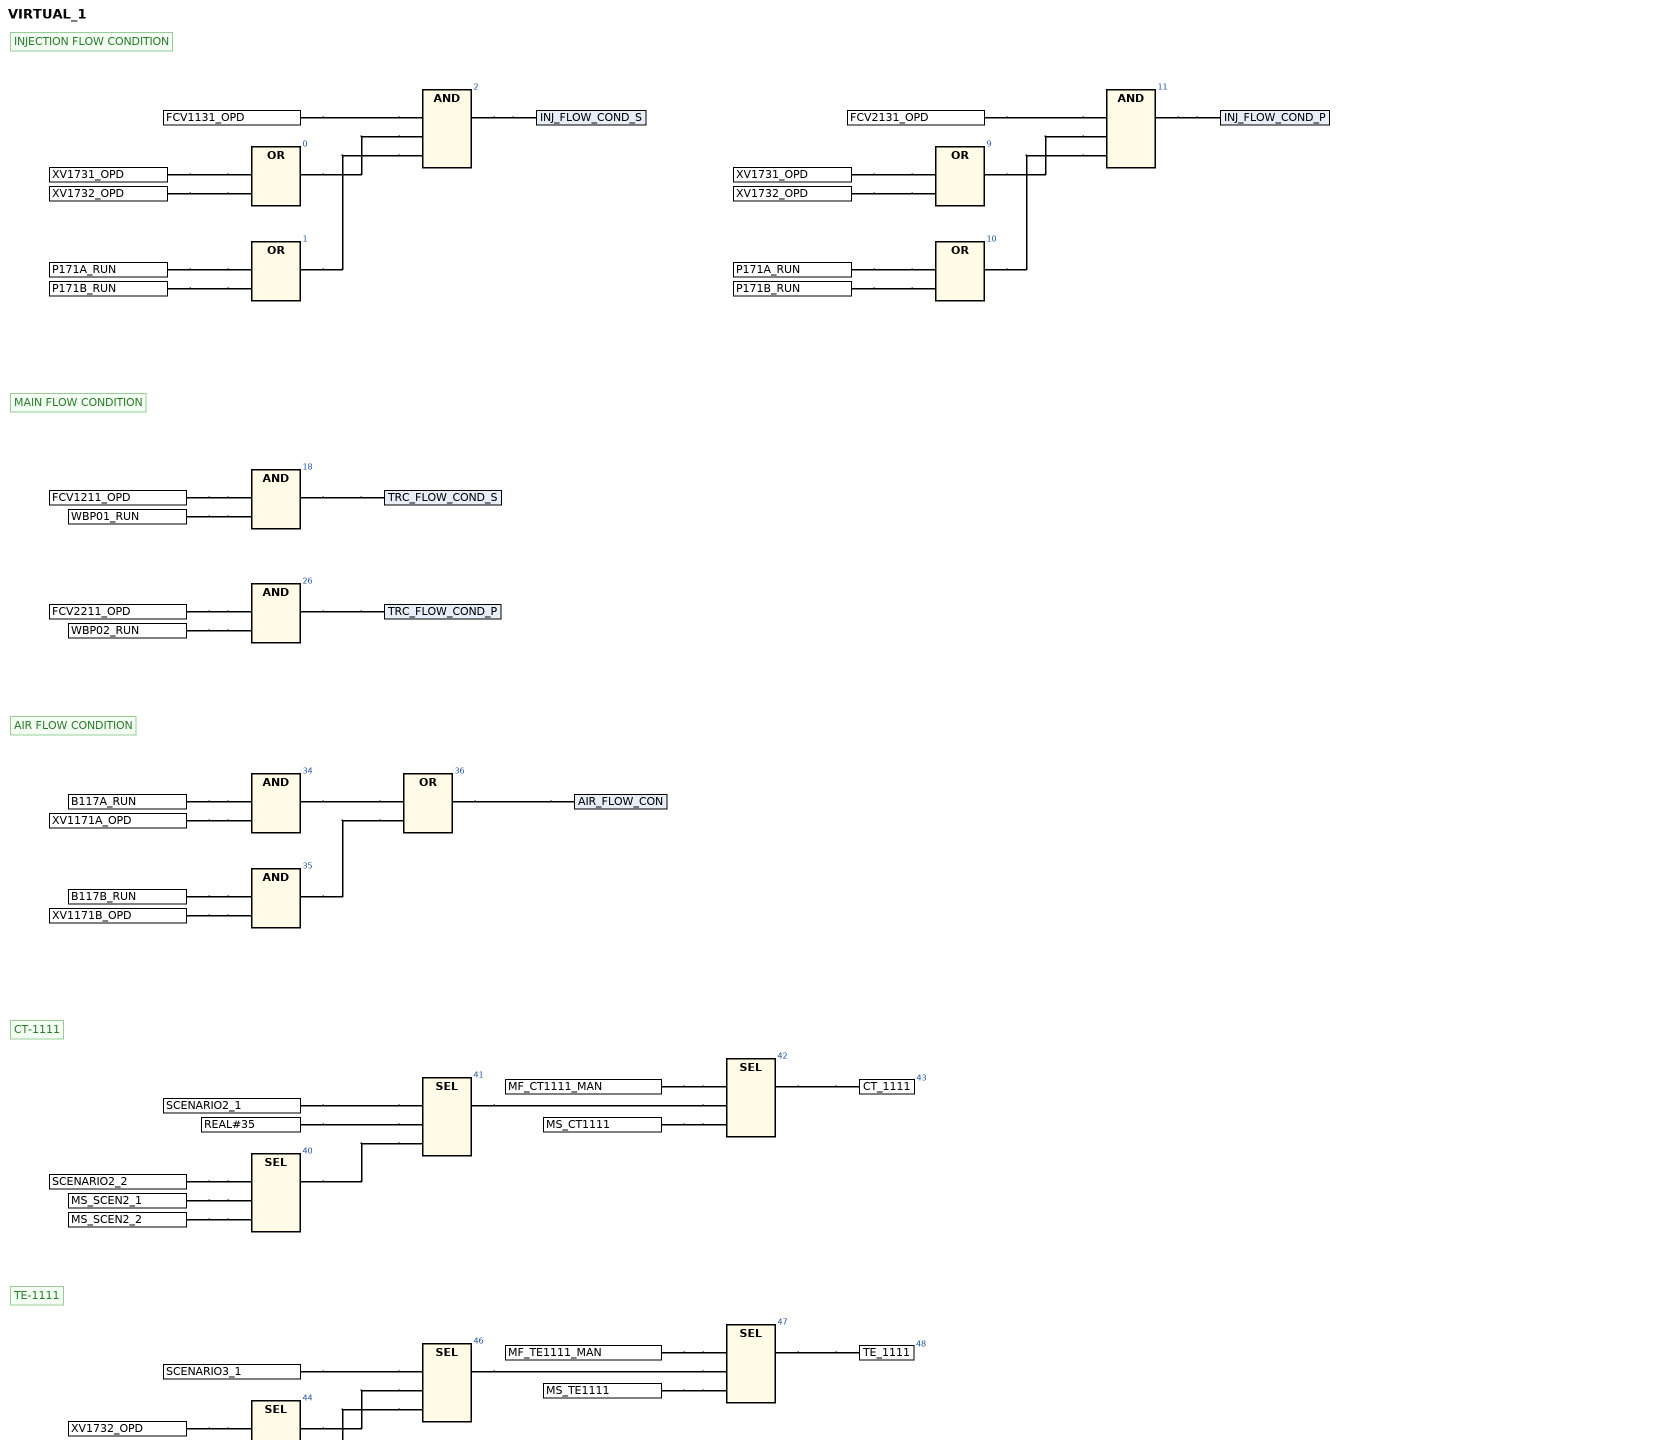
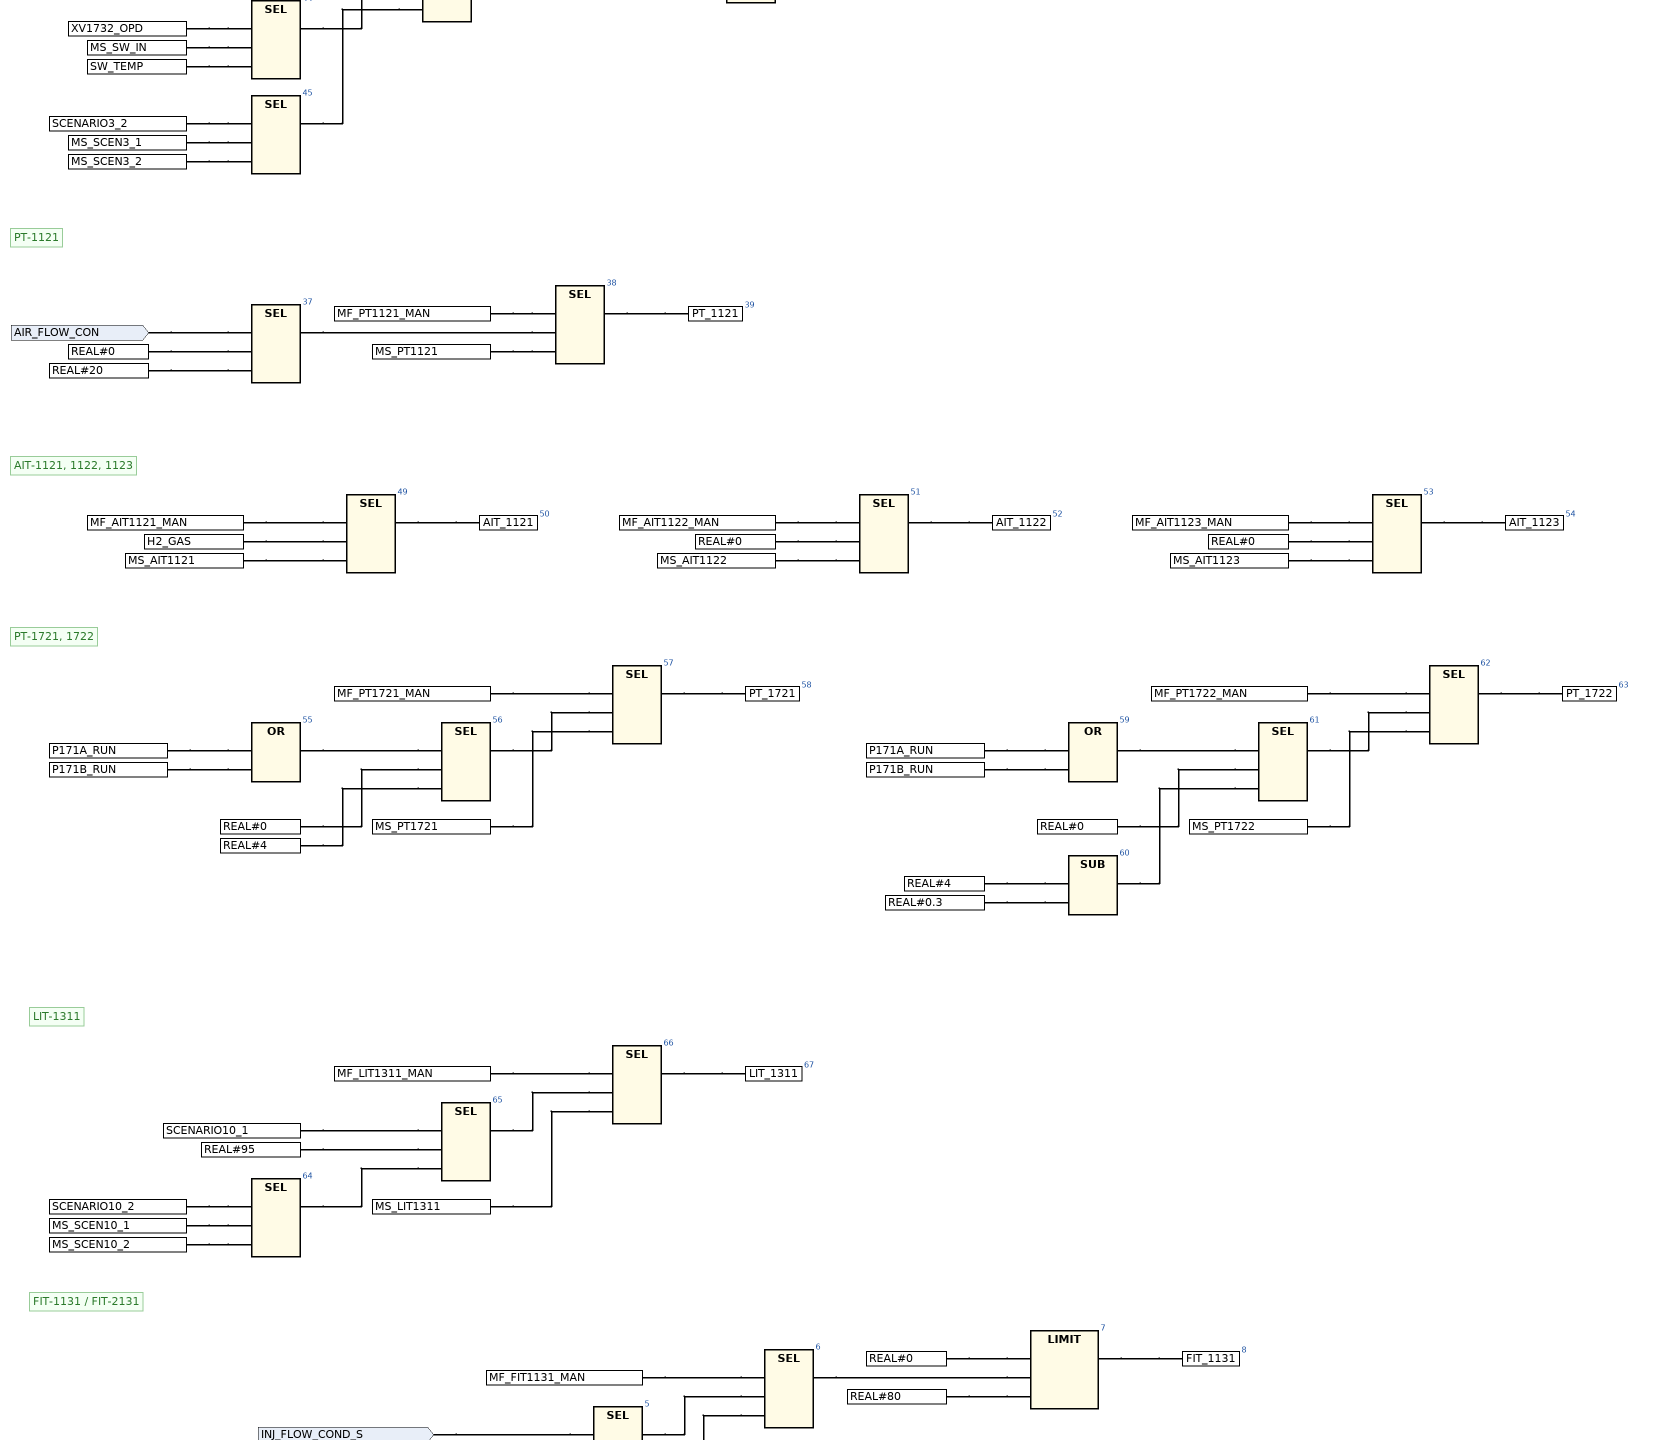
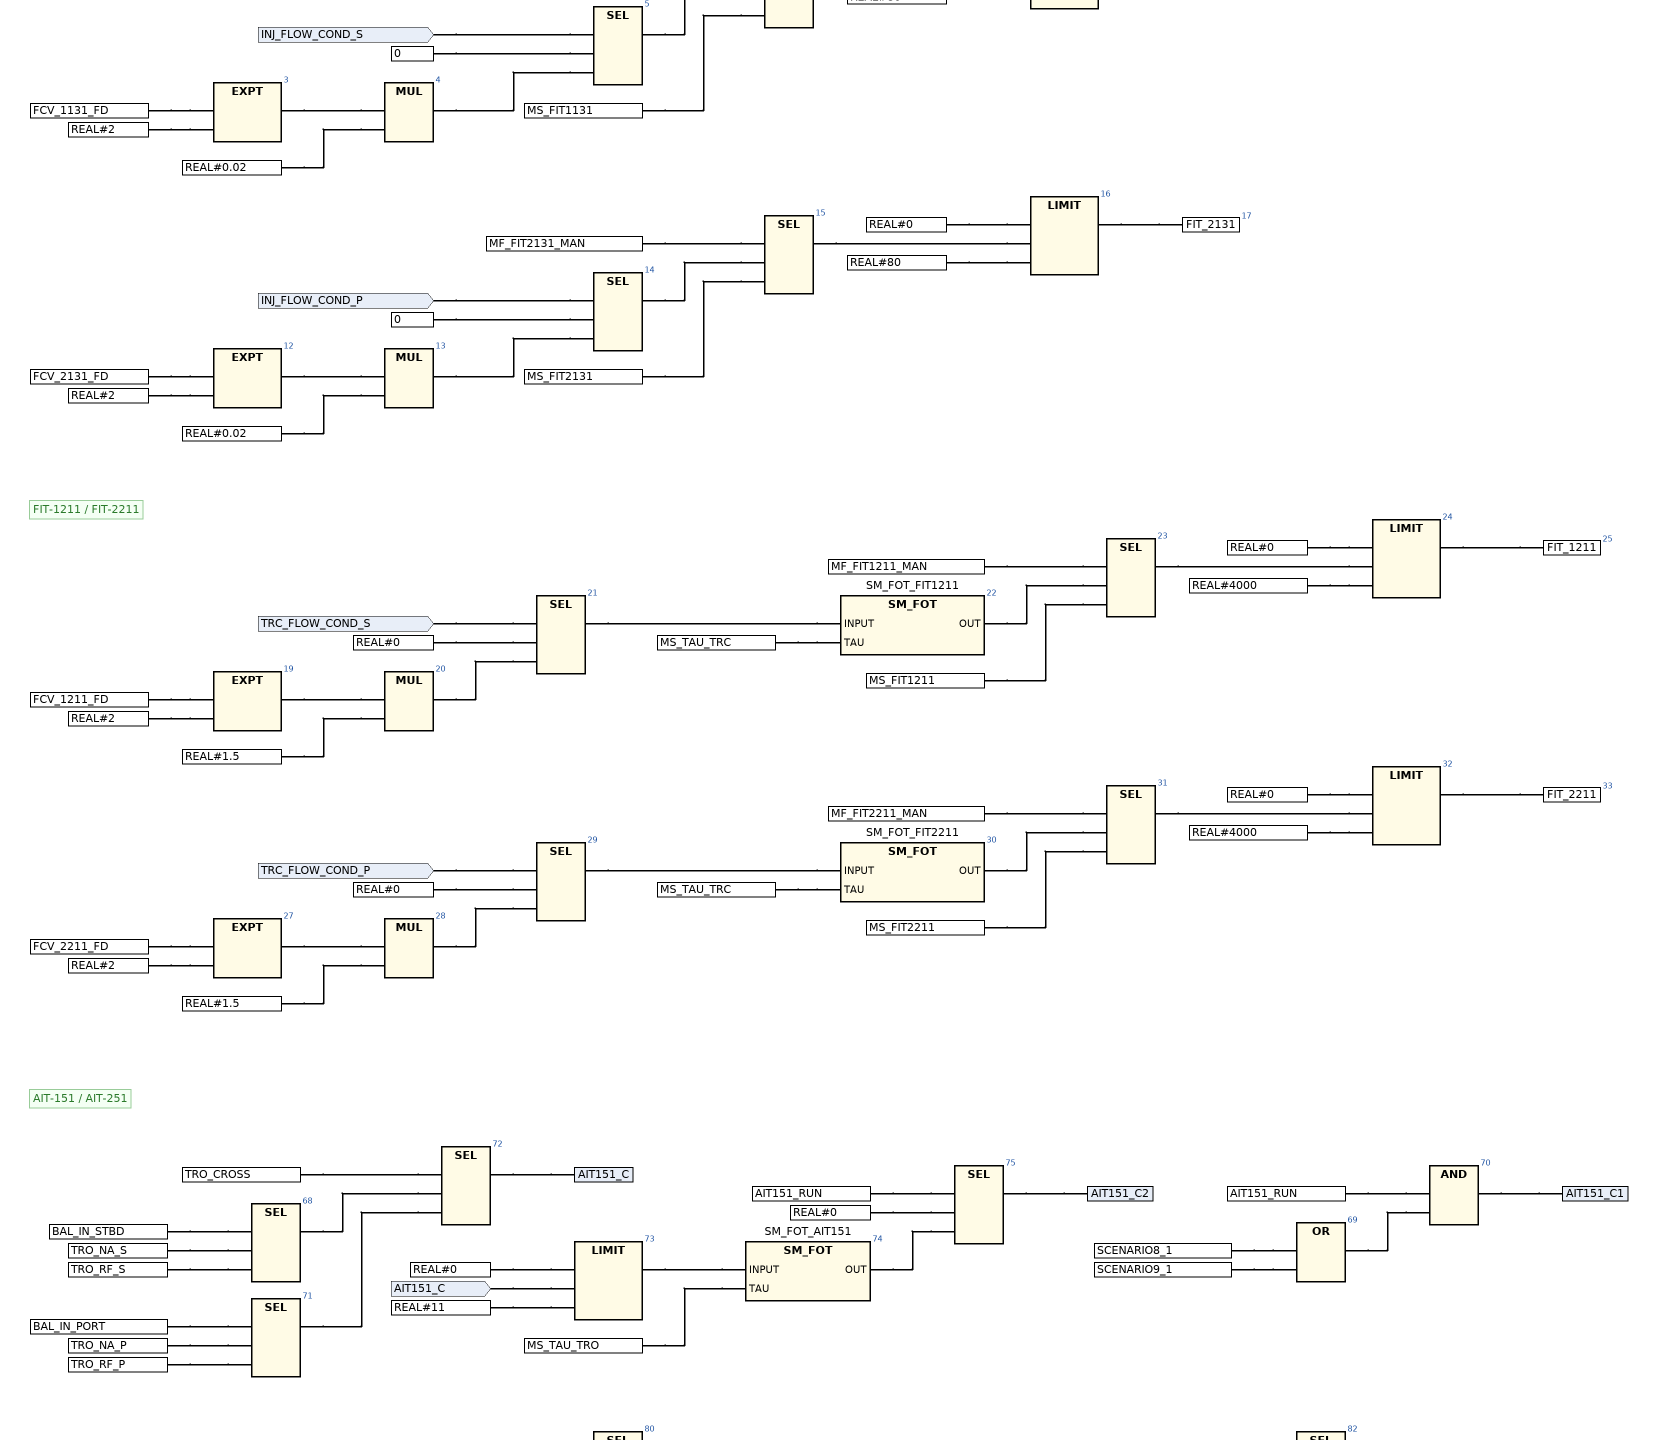
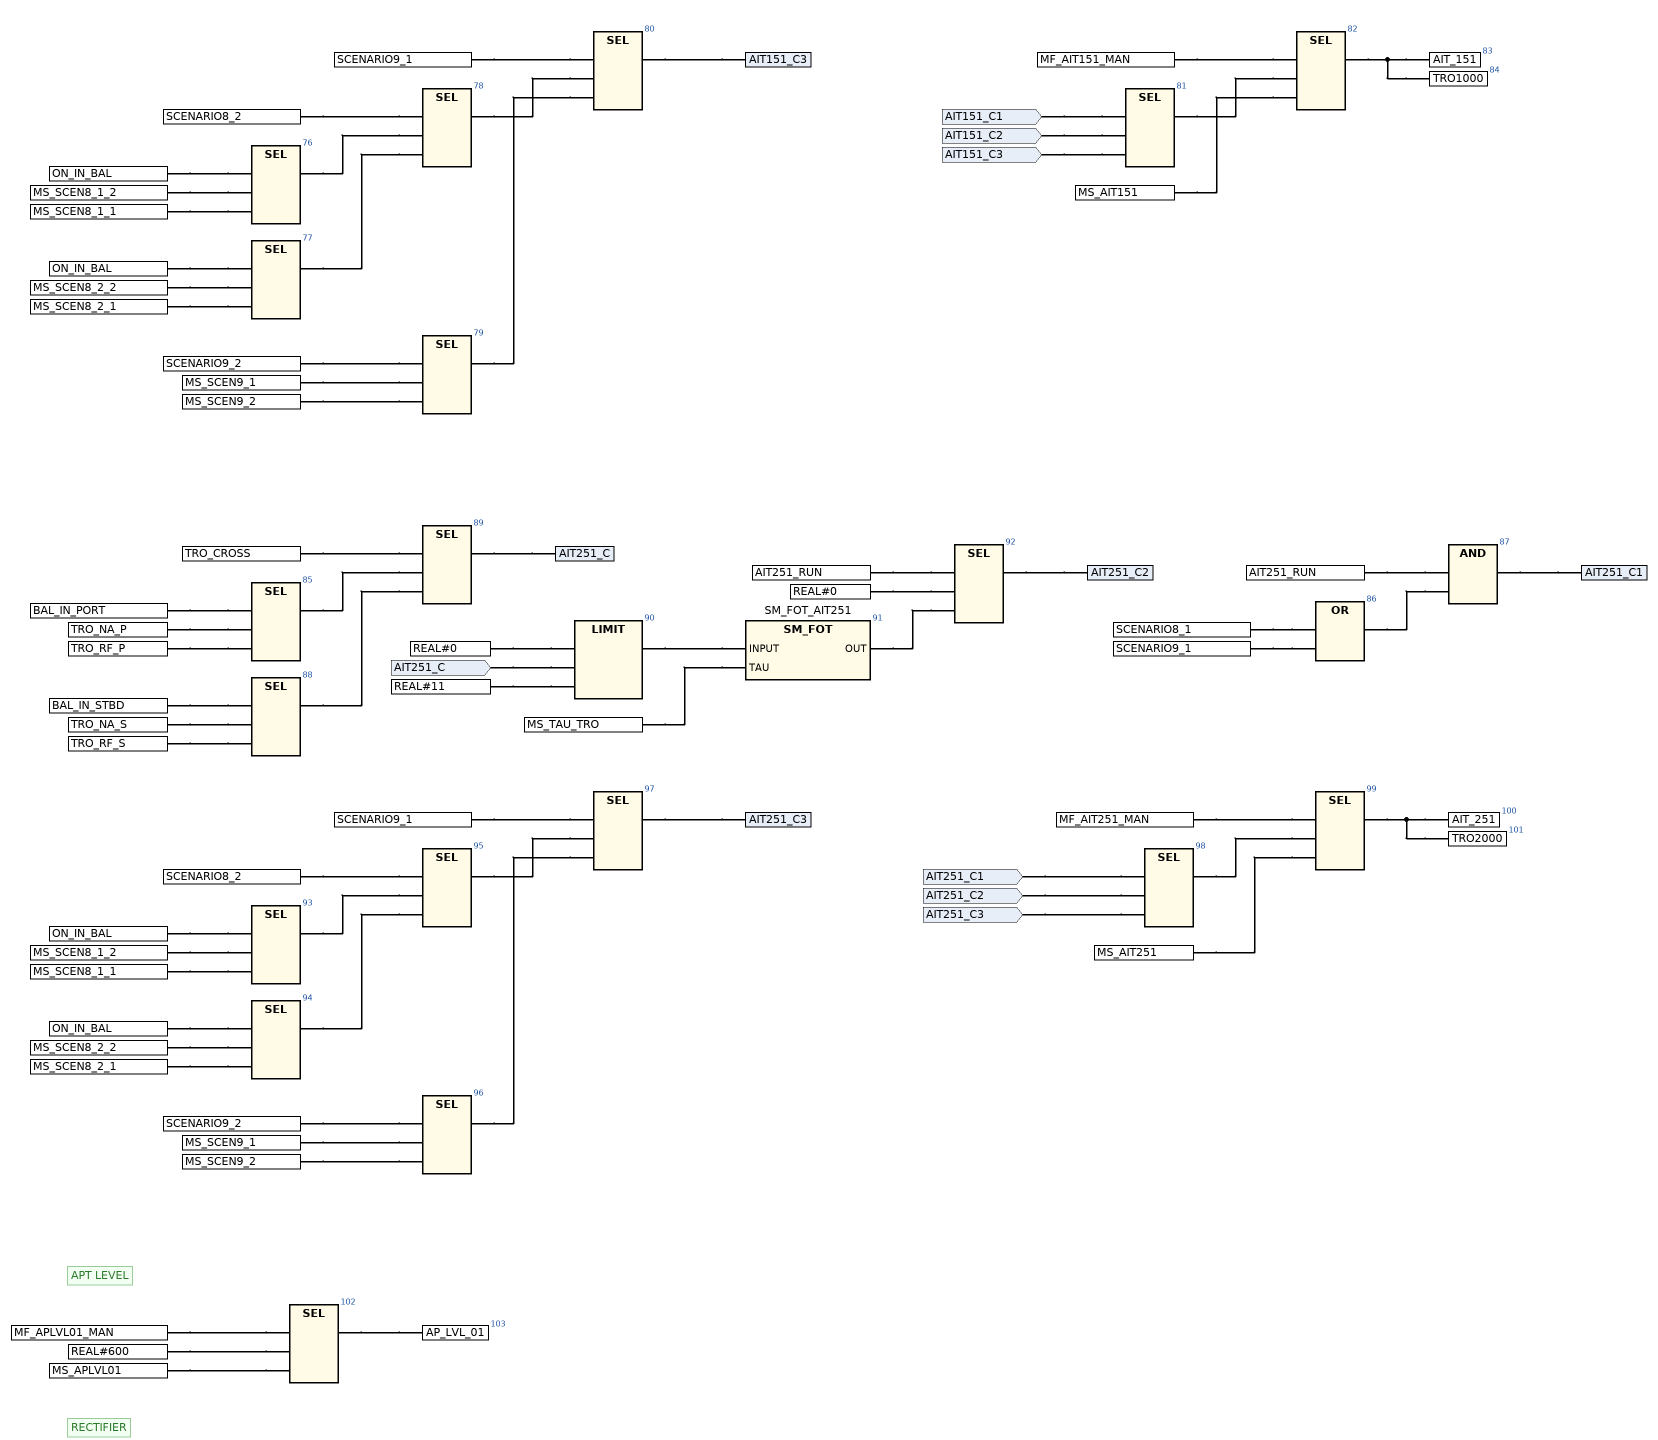
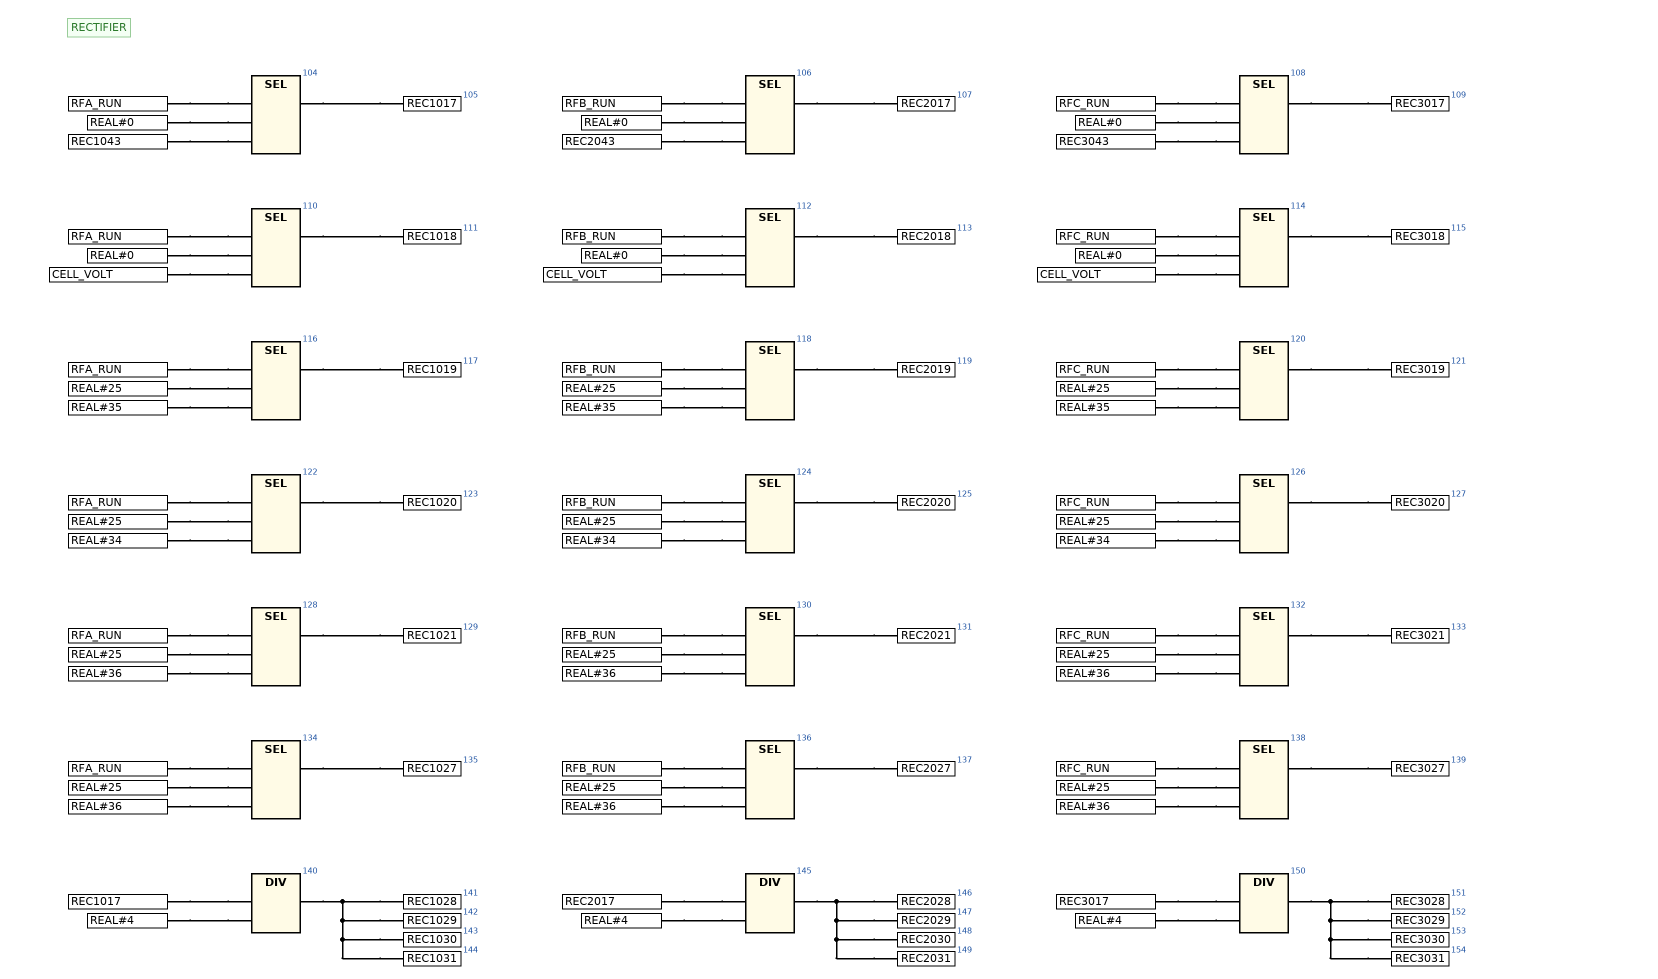
// INJECTION FLOW CONDITION
(* FCV1131_OPD AND (XV1731_OPD OR XV1732_OPD) AND (P171A_RUN OR P171B_RUN); result not used *)
// FIT-1131 / FIT-2131
FIT_1131 := LIMIT(REAL#0, SEL(MF_FIT1131_MAN, SEL(_w1, 0, EXPT(FCV_1131_FD, REAL#2) * REAL#0.02), MS_FIT1131), REAL#80);
(* FCV2131_OPD AND (XV1731_OPD OR XV1732_OPD) AND (P171A_RUN OR P171B_RUN); result not used *)
FIT_2131 := LIMIT(REAL#0, SEL(MF_FIT2131_MAN, SEL(_w2, 0, EXPT(FCV_2131_FD, REAL#2) * REAL#0.02), MS_FIT2131), REAL#80);
// MAIN FLOW CONDITION
(* FCV1211_OPD AND WBP01_RUN; result not used *)
// FIT-1211 / FIT-2211
SM_FOT_FIT1211(INPUT := SEL(_w3, REAL#0, EXPT(FCV_1211_FD, REAL#2) * REAL#1.5), TAU := MS_TAU_TRC); // SM_FOT
FIT_1211 := LIMIT(REAL#0, SEL(MF_FIT1211_MAN, SM_FOT_FIT1211.OUT, MS_FIT1211), REAL#4000);
(* FCV2211_OPD AND WBP02_RUN; result not used *)
SM_FOT_FIT2211(INPUT := SEL(_w4, REAL#0, EXPT(FCV_2211_FD, REAL#2) * REAL#1.5), TAU := MS_TAU_TRC); // SM_FOT
FIT_2211 := LIMIT(REAL#0, SEL(MF_FIT2211_MAN, SM_FOT_FIT2211.OUT, MS_FIT2211), REAL#4000);
// AIR FLOW CONDITION
(* B117A_RUN AND XV1171A_OPD OR B117B_RUN AND XV1171B_OPD; result not used *)
// PT-1121
PT_1121 := SEL(MF_PT1121_MAN, SEL(_w5, REAL#0, REAL#20), MS_PT1121);
// CT-1111
CT_1111 := SEL(MF_CT1111_MAN, SEL(SCENARIO2_1, REAL#35, SEL(SCENARIO2_2, MS_SCEN2_1, MS_SCEN2_2)), MS_CT1111);
// TE-1111
TE_1111 := SEL(MF_TE1111_MAN, SEL(SCENARIO3_1, SEL(XV1732_OPD, MS_SW_IN, SW_TEMP), SEL(SCENARIO3_2, MS_SCEN3_1, MS_SCEN3_2)), MS_TE1111);
// AIT-1121, 1122, 1123
AIT_1121 := SEL(MF_AIT1121_MAN, H2_GAS, MS_AIT1121);
AIT_1122 := SEL(MF_AIT1122_MAN, REAL#0, MS_AIT1122);
AIT_1123 := SEL(MF_AIT1123_MAN, REAL#0, MS_AIT1123);
// PT-1721, 1722
PT_1721 := SEL(MF_PT1721_MAN, SEL(P171A_RUN OR P171B_RUN, REAL#0, REAL#4), MS_PT1721);
PT_1722 := SEL(MF_PT1722_MAN, SEL(P171A_RUN OR P171B_RUN, REAL#0, REAL#4 - REAL#0.3), MS_PT1722);
// LIT-1311
LIT_1311 := SEL(MF_LIT1311_MAN, SEL(SCENARIO10_1, REAL#95, SEL(SCENARIO10_2, MS_SCEN10_1, MS_SCEN10_2)), MS_LIT1311);
// AIT-151 / AIT-251
(* AIT151_RUN AND (SCENARIO8_1 OR SCENARIO9_1); result not used *)
(* SEL(TRO_CROSS, SEL(BAL_IN_STBD, TRO_NA_S, TRO_RF_S), SEL(BAL_IN_PORT, TRO_NA_P, TRO_RF_P)); result not used *)
SM_FOT_AIT151(INPUT := LIMIT(REAL#0, _w6, REAL#11), TAU := MS_TAU_TRO); // SM_FOT
(* SEL(AIT151_RUN, REAL#0, SM_FOT_AIT151.OUT); result not used *)
(* SEL(SCENARIO9_1, SEL(SCENARIO8_2, SEL(ON_IN_BAL, MS_SCEN8_1_2, MS_SCEN8_1_1), SEL(ON_IN_BAL, MS_SCEN8_2_2, MS_SCEN8_2_1)), SEL(SCENARIO9_2, MS_SCEN9_1, MS_SCEN9_2)); result not used *)
_w10 := SEL(MF_AIT151_MAN, SEL(_w7, _w8, _w9), MS_AIT151);
AIT_151 := _w10;
TRO1000 := _w10;
(* AIT251_RUN AND (SCENARIO8_1 OR SCENARIO9_1); result not used *)
(* SEL(TRO_CROSS, SEL(BAL_IN_PORT, TRO_NA_P, TRO_RF_P), SEL(BAL_IN_STBD, TRO_NA_S, TRO_RF_S)); result not used *)
SM_FOT_AIT251(INPUT := LIMIT(REAL#0, _w11, REAL#11), TAU := MS_TAU_TRO); // SM_FOT
(* SEL(AIT251_RUN, REAL#0, SM_FOT_AIT251.OUT); result not used *)
(* SEL(SCENARIO9_1, SEL(SCENARIO8_2, SEL(ON_IN_BAL, MS_SCEN8_1_2, MS_SCEN8_1_1), SEL(ON_IN_BAL, MS_SCEN8_2_2, MS_SCEN8_2_1)), SEL(SCENARIO9_2, MS_SCEN9_1, MS_SCEN9_2)); result not used *)
_w15 := SEL(MF_AIT251_MAN, SEL(_w12, _w13, _w14), MS_AIT251);
AIT_251 := _w15;
TRO2000 := _w15;
// APT LEVEL
AP_LVL_01 := SEL(MF_APLVL01_MAN, REAL#600, MS_APLVL01);
// RECTIFIER
REC1017 := SEL(RFA_RUN, REAL#0, REC1043);
REC2017 := SEL(RFB_RUN, REAL#0, REC2043);
REC3017 := SEL(RFC_RUN, REAL#0, REC3043);
REC1018 := SEL(RFA_RUN, REAL#0, CELL_VOLT);
REC2018 := SEL(RFB_RUN, REAL#0, CELL_VOLT);
REC3018 := SEL(RFC_RUN, REAL#0, CELL_VOLT);
REC1019 := SEL(RFA_RUN, REAL#25, REAL#35);
REC2019 := SEL(RFB_RUN, REAL#25, REAL#35);
REC3019 := SEL(RFC_RUN, REAL#25, REAL#35);
REC1020 := SEL(RFA_RUN, REAL#25, REAL#34);
REC2020 := SEL(RFB_RUN, REAL#25, REAL#34);
REC3020 := SEL(RFC_RUN, REAL#25, REAL#34);
REC1021 := SEL(RFA_RUN, REAL#25, REAL#36);
REC2021 := SEL(RFB_RUN, REAL#25, REAL#36);
REC3021 := SEL(RFC_RUN, REAL#25, REAL#36);
REC1027 := SEL(RFA_RUN, REAL#25, REAL#36);
REC2027 := SEL(RFB_RUN, REAL#25, REAL#36);
REC3027 := SEL(RFC_RUN, REAL#25, REAL#36);
_w16 := REC1017 / REAL#4;
REC1028 := _w16;
REC1029 := _w16;
REC1030 := _w16;
REC1031 := _w16;
_w17 := REC2017 / REAL#4;
REC2028 := _w17;
REC2029 := _w17;
REC2030 := _w17;
REC2031 := _w17;
_w18 := REC3017 / REAL#4;
REC3028 := _w18;
REC3029 := _w18;
REC3030 := _w18;
REC3031 := _w18;

END_PROGRAM

// Device/Application/Logic/0.SIMULATION FBD/SM_FOT
FUNCTION_BLOCK SM_FOT
VAR_INPUT
	INPUT : REAL;
	TAU : REAL := 0.5;				// TIME CONSTANT (0~1)
END_VAR
VAR_OUTPUT
	OUT : REAL;
END_VAR
VAR
	Y1 : REAL;				//EXISTING VALUE
	Y2 : REAL;				//VALUE AFTER CHANGE
	ET_0 : TON;				//ELAPSED TIME AFTER VALUE CHANGE
	INTEGRAL_ET: INTEGRAL;
	TP_0: TP;
END_VAR
VAR // added by the converter: edge detectors and wires of the graphical bodies
    _w1, _w6 : REAL;
    _w2, _w5 : BOOL;
    _w3, _w4, _w7, _w8 : ANY;
END_VAR

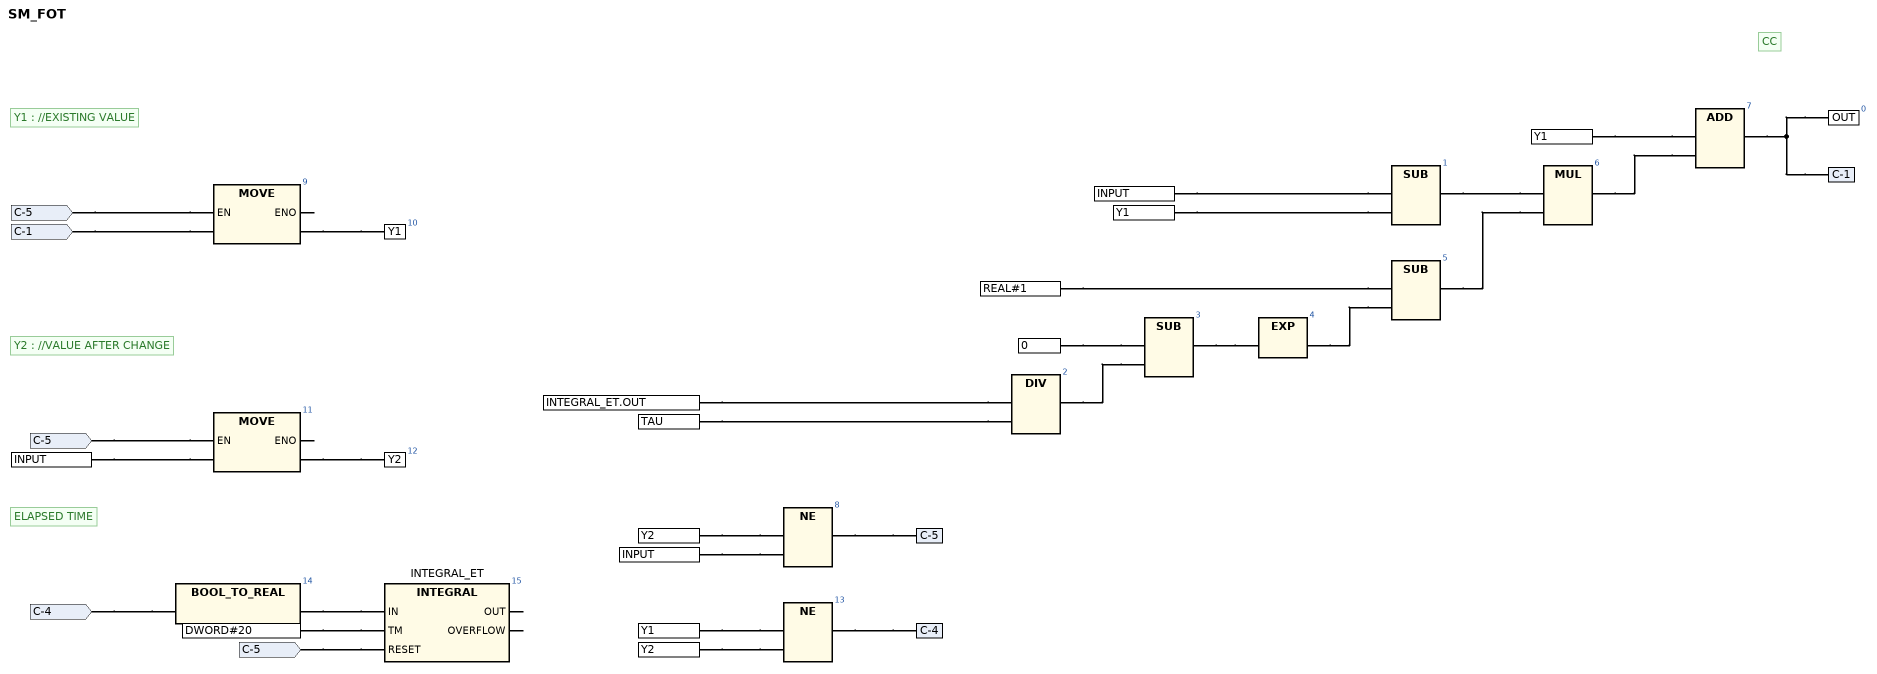
OUT := _w1;
// CC
_w1 := Y1 + (INPUT - Y1) * (REAL#1 - EXP(0 - INTEGRAL_ET.OUT / TAU));
(* Y2 <> INPUT; result not used *)
// Y1 : //EXISTING VALUE
IF _w2 THEN _w4 := _w3; END_IF
Y1 := _w4;
// Y2 : //VALUE AFTER CHANGE
IF _w5 THEN _w6 := INPUT; END_IF
Y2 := _w6;
(* Y1 <> Y2; result not used *)
// ELAPSED TIME
INTEGRAL_ET(IN := BOOL_TO_REAL(_w7), TM := DWORD#20, RESET := _w8); // INTEGRAL

END_FUNCTION_BLOCK

// Device/Application/Logic/0.SIMULATION/VIRTUAL_2
PROGRAM VIRTUAL_2
VAR
END_VAR

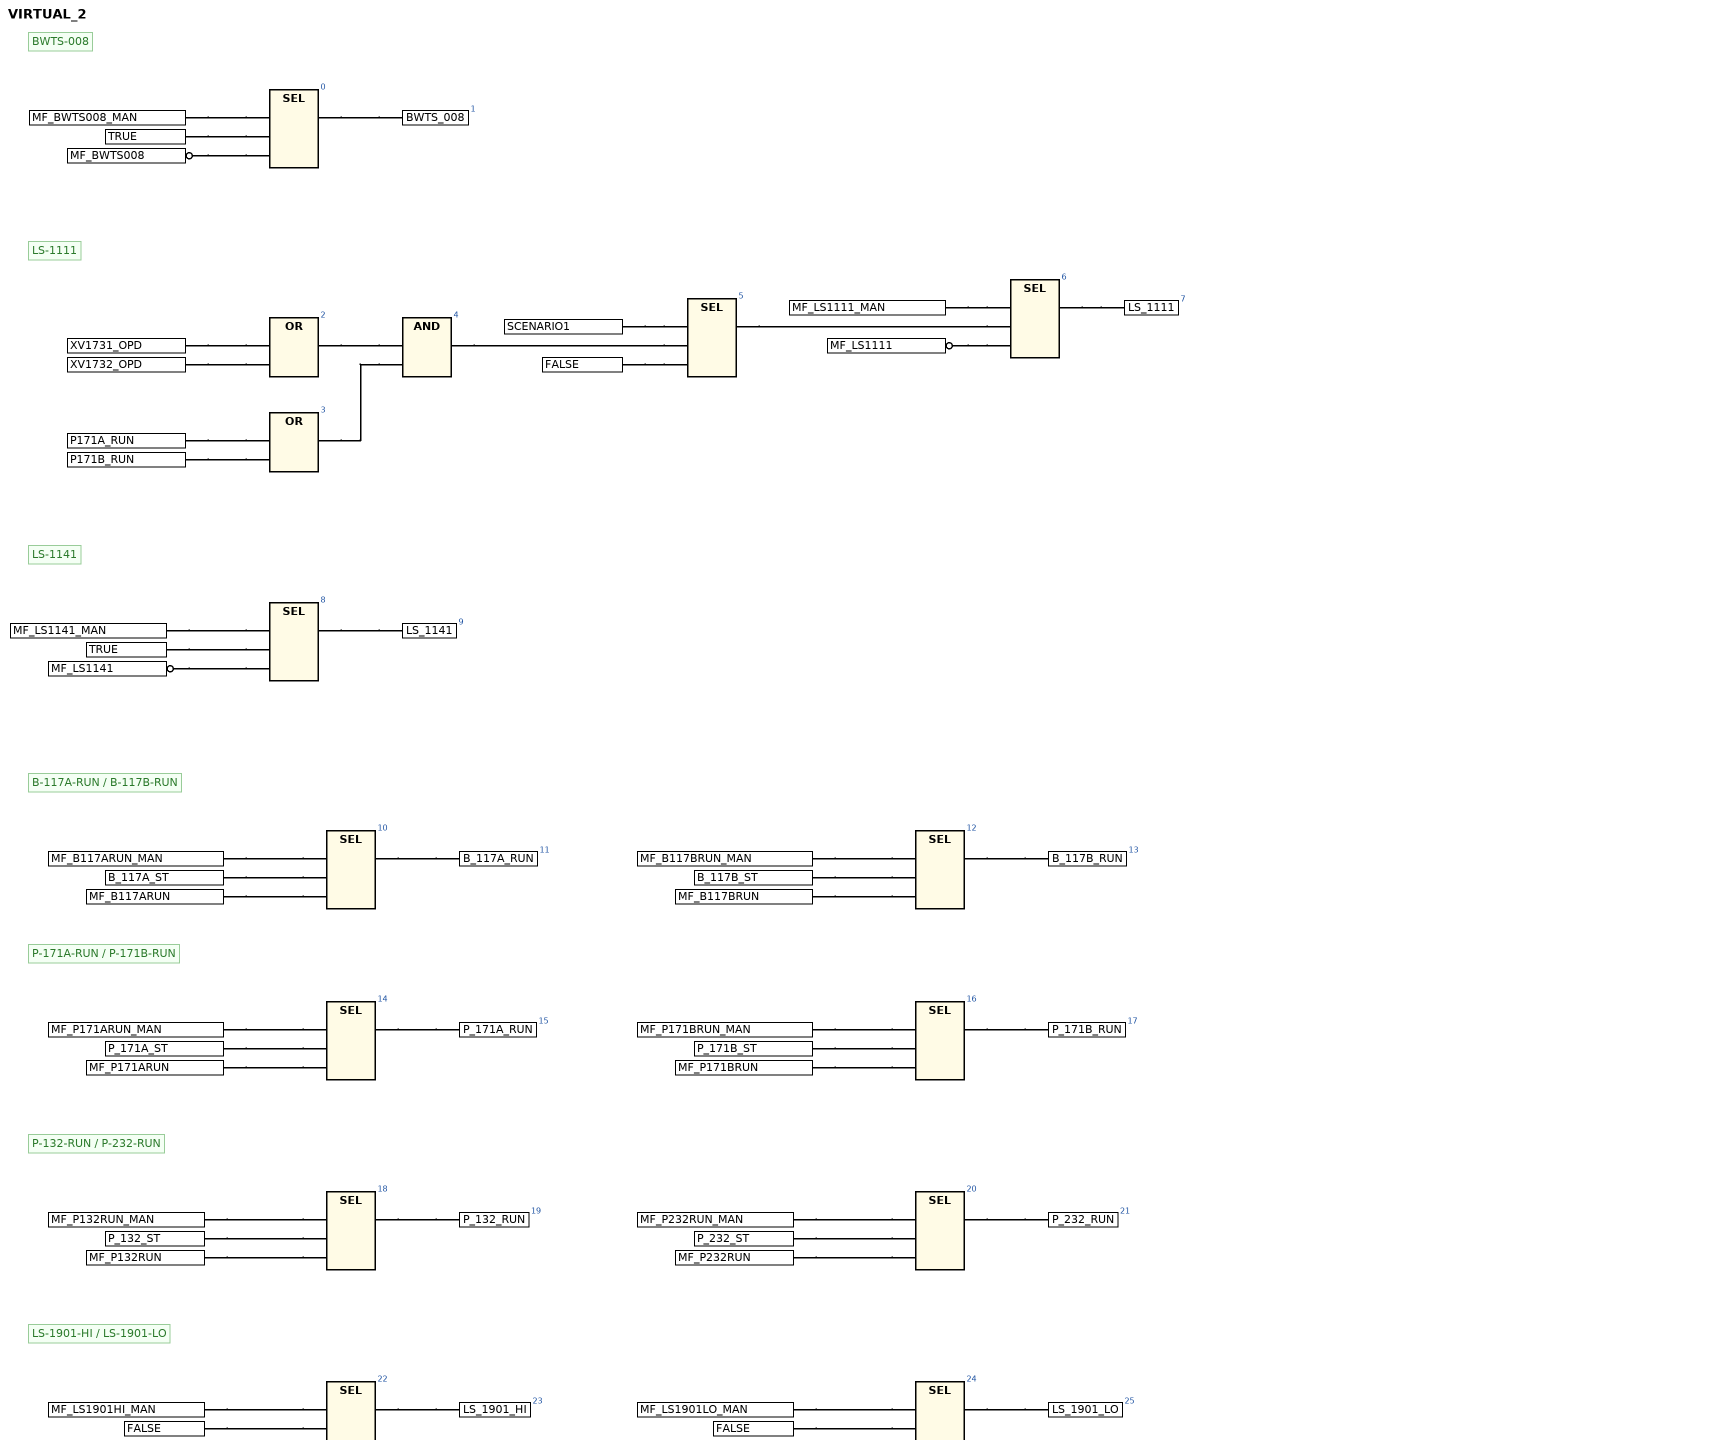
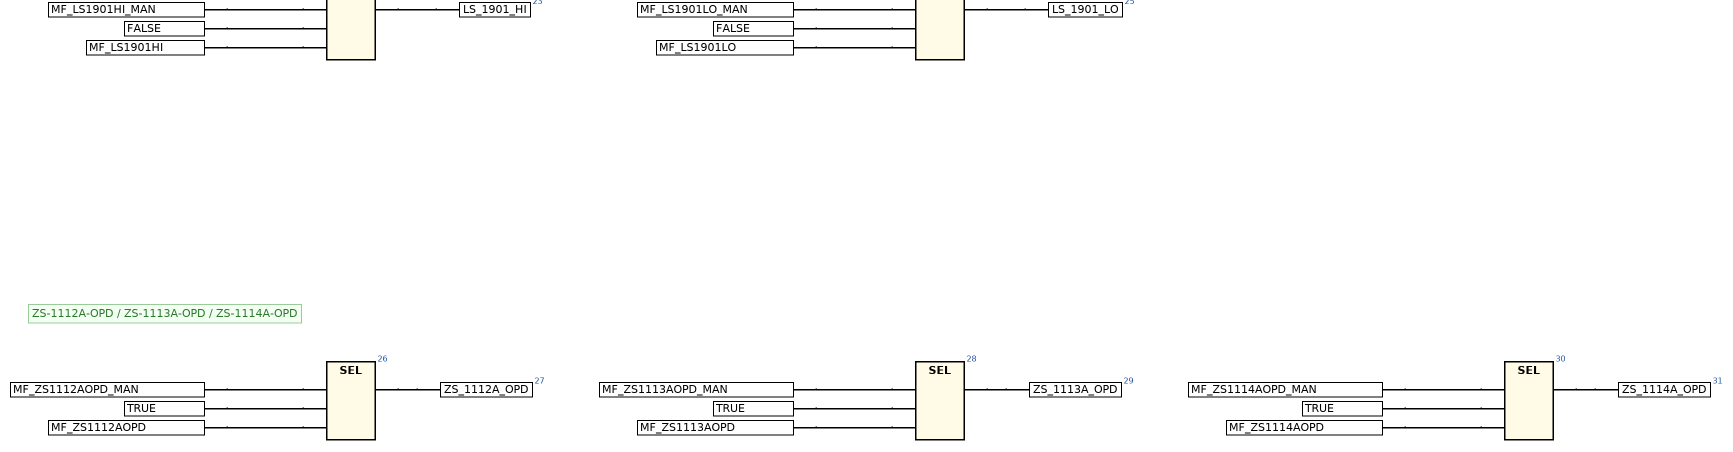
// BWTS-008
BWTS_008 := SEL(MF_BWTS008_MAN, TRUE, NOT MF_BWTS008);
// LS-1111
LS_1111 := SEL(MF_LS1111_MAN, SEL(SCENARIO1, (XV1731_OPD OR XV1732_OPD) AND (P171A_RUN OR P171B_RUN), FALSE), NOT MF_LS1111);
// LS-1141
LS_1141 := SEL(MF_LS1141_MAN, TRUE, NOT MF_LS1141);
// B-117A-RUN / B-117B-RUN
B_117A_RUN := SEL(MF_B117ARUN_MAN, B_117A_ST, MF_B117ARUN);
B_117B_RUN := SEL(MF_B117BRUN_MAN, B_117B_ST, MF_B117BRUN);
// P-171A-RUN / P-171B-RUN
P_171A_RUN := SEL(MF_P171ARUN_MAN, P_171A_ST, MF_P171ARUN);
P_171B_RUN := SEL(MF_P171BRUN_MAN, P_171B_ST, MF_P171BRUN);
// P-132-RUN / P-232-RUN
P_132_RUN := SEL(MF_P132RUN_MAN, P_132_ST, MF_P132RUN);
P_232_RUN := SEL(MF_P232RUN_MAN, P_232_ST, MF_P232RUN);
// LS-1901-HI / LS-1901-LO
LS_1901_HI := SEL(MF_LS1901HI_MAN, FALSE, MF_LS1901HI);
LS_1901_LO := SEL(MF_LS1901LO_MAN, FALSE, MF_LS1901LO);
// ZS-1112A-OPD / ZS-1113A-OPD / ZS-1114A-OPD
ZS_1112A_OPD := SEL(MF_ZS1112AOPD_MAN, TRUE, MF_ZS1112AOPD);
ZS_1113A_OPD := SEL(MF_ZS1113AOPD_MAN, TRUE, MF_ZS1113AOPD);
ZS_1114A_OPD := SEL(MF_ZS1114AOPD_MAN, TRUE, MF_ZS1114AOPD);

END_PROGRAM

// Device/Application/Logic/0.SIMULATION/VIRTUAL_3
PROGRAM VIRTUAL_3
VAR

END_VAR

XV_1171A_OPD := XV_1171A_CMD;
XV_1171A_CLD := NOT XV_1171A_CMD;
XV_1171B_OPD := XV_1171B_CMD;
XV_1171B_CLD := NOT XV_1171B_CMD;

FCV_1131_FD := FCV_1131_CMD;
FCV_2131_FD := FCV_2131_CMD;

FCV_1211_FD := FCV_1211_CMD;
FCV_2211_FD := FCV_2211_CMD;

P_132_FD := P_132_CMD;
P_232_FD := P_232_CMD;

REC1000 := RF_142A_ST;
REC2000 := RF_142B_ST;
REC3000 := RF_142C_ST;

END_PROGRAM

// Device/Application/Logic/0.SIMULATION FBD/SM_RF_TRO1
FUNCTION_BLOCK SM_RF_TRO1
VAR_INPUT
	TOTAL_CURRENT : REAL;
	INJ_S : REAL;
	INJ_P : REAL;
	TRC_S : REAL;
	TRC_P : REAL;
END_VAR
VAR_OUTPUT
	TRO_S : REAL;
	TRO_P : REAL;
END_VAR
VAR
	CURR_EFF : REAL := 0.7;			//Current efficiency : 0~1
	FARA : REAL := 96484.55461;		//Faraday constant
	MWCL : REAL := 70.9054;			//M.W. of Chlorine
	CELL_N : REAL := 41;			//No. of cell 
	CURR_T : REAL;					//Total currunt
	CLPROD : REAL;
	INJ_RATIO_S : REAL;
	INJ_RATIO_P : REAL;
END_VAR

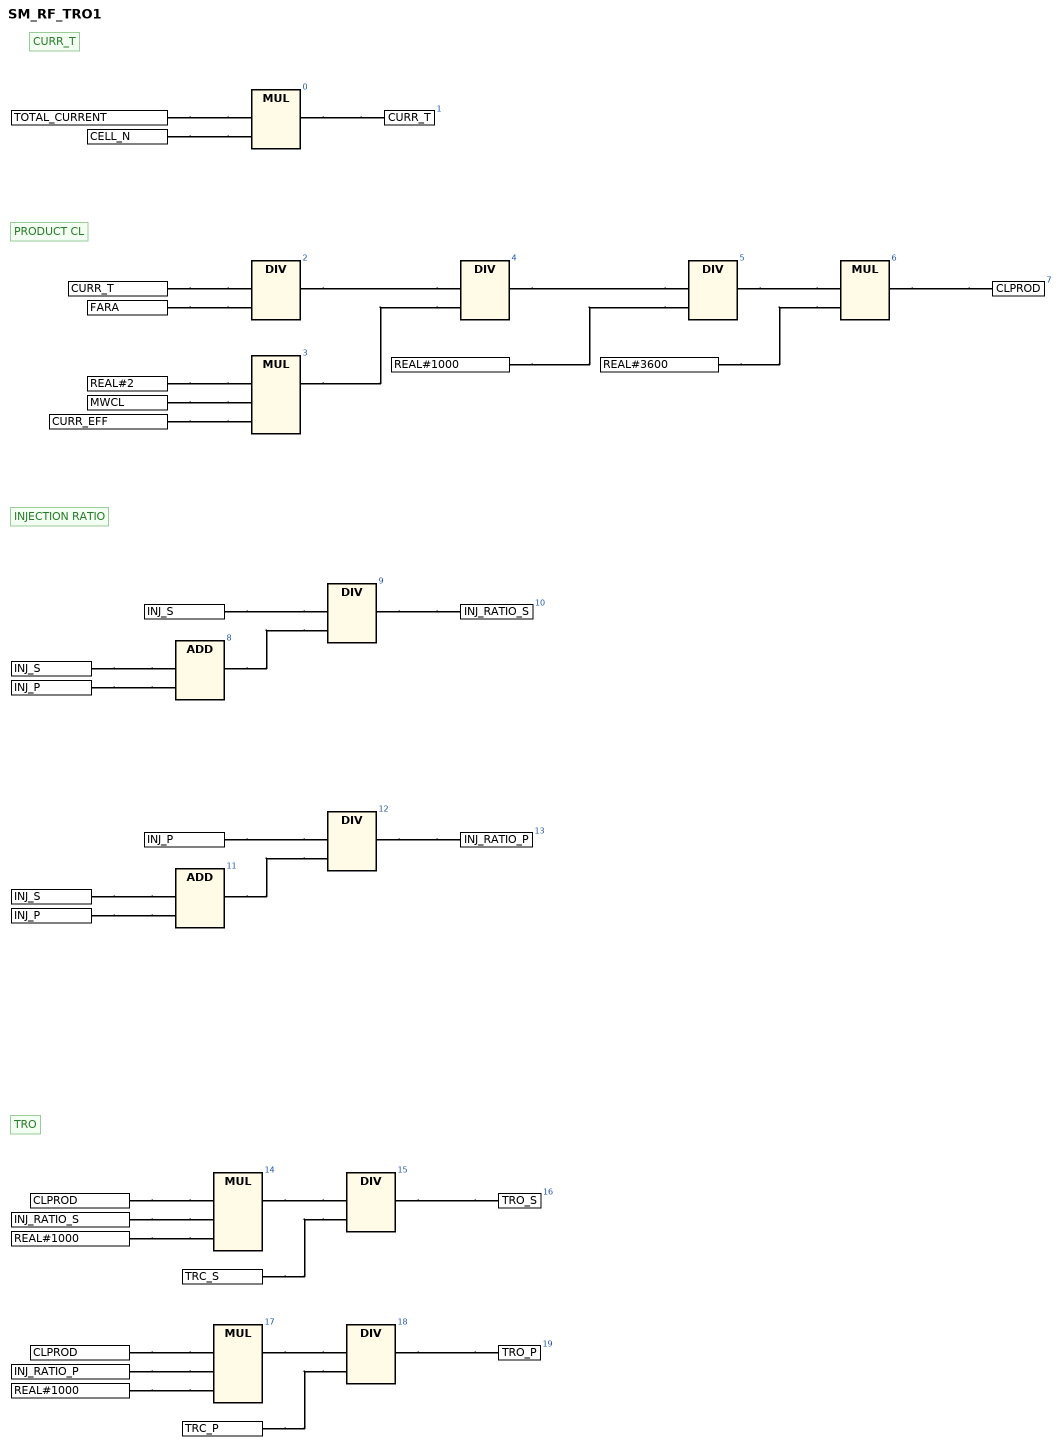
// CURR_T
CURR_T := TOTAL_CURRENT * CELL_N;
// PRODUCT CL
CLPROD := (((CURR_T / FARA) / (REAL#2 * MWCL * CURR_EFF)) / REAL#1000) * REAL#3600;
// INJECTION RATIO
INJ_RATIO_S := INJ_S / (INJ_S + INJ_P);
INJ_RATIO_P := INJ_P / (INJ_S + INJ_P);
// TRO
TRO_S := (CLPROD * INJ_RATIO_S * REAL#1000) / TRC_S;
TRO_P := (CLPROD * INJ_RATIO_P * REAL#1000) / TRC_P;

END_FUNCTION_BLOCK

// Device/Application/Logic/0.SIMULATION FBD/SM_FU_DP
FUNCTION_BLOCK SM_FU_DP
VAR_INPUT
	WQ : REAL;				//WATER QUALITY
	A0 : REAL;				//FILTRATION AREA
	FLOW_MAIN : REAL;		
	FLUSHING : BOOL;
	OPENING: BOOL;
END_VAR
VAR_OUTPUT
	OUT : REAL;
END_VAR
VAR
	K1 : REAL := 4.30E-04;
	K2 : REAL := 2.66551E-06;
	FQ : REAL;
	AC : REAL;				//CLOGGED AREA
	aa : REAL;				//Effective filtration area
	INTEGRAL_0 : INTEGRAL;
END_VAR

INTEGRAL_0(IN:= SEL(OPENING, 0, 1), TM:= DWORD#20, RESET:= FLUSHING);
FQ := FLOW_MAIN * INTEGRAL_0.OUT / 3600;
AC := K1 * WQ * FQ;
aa := A0 - AC;
OUT := K2 * EXPT(FLOW_MAIN/aa, 2);

END_FUNCTION_BLOCK
